Fanuc KAREL source: kf00047.KL

-- PROVISIONAL review KL for V1013-1; original PC SHA256 b845a61647ab4263b8c148117acdb5005c3ae877f09dc60b76ded7a8d779430a
-- Incomplete behavior may be omitted. Consult companion uncertainty JSON. Do not deploy.
PROGRAM KF00047
%NOLOCKGROUP
VAR
  I : INTEGER
  J : INTEGER
  X : REAL
  Y : REAL
  B : BOOLEAN
  C : BOOLEAN
  TXT : STRING[80]
  TXT2 : STRING[80]
  STATUS : INTEGER
-- UNRESOLVED_DECL AI type=002010
-- UNRESOLVED_DECL BI type=002010
-- UNRESOLVED_DECL P type=000102
-- UNRESOLVED_DECL JP type=000199
-- UNRESOLVED_DECL PF type=000101
-- UNRESOLVED_DECL V1 type=000013
-- UNRESOLVED_DECL V2 type=000013
BEGIN
  -- UNRESOLVED_PC offsets 5-12; opcodes 9D,23
  -- UNRESOLVED_PC offsets 17-28; opcodes 2E,23
  -- UNRESOLVED_PC offsets 33-46; opcodes 21,9D,57,79
  -- UNRESOLVED_PC offsets 51-68; opcodes 21,2E,57,79
  -- UNRESOLVED_PC offsets 73-84; opcodes 2E,23
  -- UNRESOLVED_PC offsets 99-103; opcodes 7F
END KF00047
